// TIA Portal V16 export
// export: Created 2021-05-10T12:38:58.3862422Z, ExportSetting WithDefaults, DisplayName Totally Integrated Automation Portal, DisplayVersion V16 Update 3, DisplayName TIA Portal Version Control Interface, DisplayVersion V16 Update 2, DisplayName TIA Portal Openness, DisplayVersion V16 Update 3, DisplayName STEP 7 Professional, DisplayVersion V16 Update 3, DisplayName STEP 7 Safety, DisplayVersion V16, DisplayName WinCC Professional, DisplayVersion V16 Update 3
VAR_GLOBAL   // PLC tag table "PAL_TestFC01001"
   Trap_dirFalseHigh AT %M12.0 : Bool;
   Trap_dirTrueLow AT %M12.1 : Bool;
   Trap_parFalseHigh AT %M12.2 : Bool;
   Trap_parTrueLow AT %M12.3 : Bool;
   Trap_dirCycFirstOn AT %M12.4 : Bool;
   Trap_parCycFirstOn AT %M12.5 : Bool;
   Trap_dirCycFirstCount AT %MW14 : Word;
   Trap_parCycFirstCount AT %MW16 : Word;
   Check_CycCount AT %MW1000 : Word;
END_VAR
